Universal Robots URScript: SUB_107.script

def SUB_107():
  global _hidden_verificationVariable=0
  set_safety_mode_transition_hardness(1)
  set_tcp(p[0.0,0.09,0.42,0.0,0.0,0.0])
  set_target_payload(0.100000, [0.135000, 0.000000, 0.225000], [10.000000, 10.000000, 10.000000, 0.000000, 0.000000, 0.000000])
  set_gravity([0.0, 0.0, 9.82])
  set_standard_analog_input_domain(0, 1)
  set_standard_analog_input_domain(1, 1)
  set_tool_analog_input_domain(0, 1)
  set_tool_analog_input_domain(1, 1)
  set_analog_outputdomain(0, 0)
  set_analog_outputdomain(1, 0)
  set_input_actions_to_default()
  set_runstate_gp_boolean_output_to_value(0, 3)
  set_tool_communication(False, 115200, 0, 1, 1.5, 3.5)
  set_tool_output_mode(0)
  set_tool_digital_output_mode(0, 1)
  set_tool_digital_output_mode(1, 1)
  set_tool_voltage(0)
  global DistPillar=-0.10159
  global CandCnt=2
  global ReCaptZ=0.05
  global port=3000
  global socket_timeout=120
  global host="192.168.1.2"
  global is_popup=False
  global pBucket=[p[0.83653, 0.40397, 0.34225, 0, 0, -1.59904], p[-0.75609, -0.54132, 0.33714, 0, -0, 1.55997], p[0, 0, 0, 0, 0, 0]]
  global CaptStepZ=0.08
  global CaptIndex=[2, 0, 0]
  global pBucketM=p[-0.76064, -0.49997, 0.35503, 0, 0, 1.57135]
  global socket_name="vt"
  global rovi_err=0
  global SubPrgResult=100
  global CurrPos=p[-0.0041, -0.42062, 0.52846, -0.0222, -3.14131, -0.00178]
  global CurrPos_p=p[-0.00291, -0.33016, 0.10856, -0.0222, -3.14131, -0.00178]
  global ForceStartZ=0.39943
  global CutOffZ=0.26446
  global Sub3100_ZMax=0.74
  global ForceStartX=-0.90368
  global Sub3100_aRot=0.2
  global Sub3100_d=0.3
  global Sub3100_Option=38
  global Sub3100_a=0.2
  global Sub3100_XdV=0.1
  global Sub3100_XdRot=8
  global ZoneDistTh=0.05
  global BucketWidth=0.95
  global ZoneBucketGap=0
  global ZoneHomeX=0.2
  global UnloadZ=0.072
  global CaptPos=p[0.757, -0.42592, -0.06353, 3.14138, 0.03448, 0.00005]
  global BucketUpperPos=p[0.471, -0.42592, -0.06353, 3.14138, 0.03448, 0.00005]
  global Sub3100_GPII18=38
  global Zone6ThX=0.1
  global Zone6ThY=0.05
  global pCV=p[-0.00039, 0.00199, -0.01591, -0.0138, 0.00523, 0.00624]
  global CaptRowNo=5
  global CrankDepthFull=0.025
  global CrankDepth=0.12406
  global Y1=[2, -101.58556, 16.83588, 47.62585]
  global Y2=p[0.20537, -0.59585, -0.22377, -0.01856, -0.01958, 1.59883]
  global EvacRadiusTh=0.3
  global EvacXTh=[-0.5, 0.5]
  global EvacYTh=[-0.8, 1]
  global EvacZTh=[-0.1, 5]
  global WorkPosNo=0
  global Zone1ZTh=0.1
  global ReCaptNo=0
  global DistPillarBak=-0.10159
  global CaptIndexWk=2
  global PoseSub=p[0, 0, 0, -0.04215, -0.01806, 0]
  global PoseAdd=p[0.26591, -0.96698, -0.01503, 2.15596, 2.2396, -0.0019]
  global RZTh=15
  global pBucketC=p[0.45, -0.8, 0.35, 0, 0, 3.1415]
  global ReCaptZWk=0
  global CheckMST=1
  global RZSub=3.31201
  global DistPillarCOTh=0.16
  global DistPillarAPTh=0.26
  global CutOffZAdd=0.24763
  global CutOffZDef=0.09
  global Y8=0
  global BKWidth_Value=[934, 985, 0]
  global BKWidth_Name="/prepro/bucket_width"
  global LevelZ=0.01684
  global NeighborZ=0.04763
  global Currpos_p_UF0=p[0.27154, 0.19262, 0.33701, -2.25553, -2.16214, -0.02728]
  global TCPSpeed=p[0, 0, 0, 0, 0, 0]
  global Sub3100_Xd=[0, 0, -0.1, 0, 0, 0]
  global Sub3100_q=2
  global Sub3100_e=-1
  global Sub3100_t=0.5
  global IsShake=False
  global BeyondZ=0.2
  global ShakeCnt=-1
  global IsSteady_01=False
  global IsSteady_02=True
  global HandInZ=0.05
  global TCPSpeedThZ=0.0005
  global ShakeWaitSec=1
  global CutOffPos=p[0.74495, -0.05741, 0.23647, -2.14909, 2.29151, 0]
  global RelMoveZ=0.075
  global ForceFeature=p[0.83653, 0.40397, -0.05775, 0, 0, -1.59904]
  global ForceAxis=[1, 1, 1, 1, 1, 1]
  global ForceValue=[0, 0, -0.04, 0, 0, 0]
  global ForceType=2
  global ForceLimit=[0.01, 0.01, -0.02505, 0.17453, 0.17453, 0.17453]
  global ForceStep=3
  global IsBLLoad=False
  global TM_BLLoad=0.5
  global Sub104__TiltZTh=[0.25, 0.4]
  global Sub104_TiltZTh=[-0.5, 0.5]
  global BucketDef=p[0.83653, 0.40397, 0.34225, 0, 0, -1.59904]
  global ForceLimitZ=[0.015, 0.05, 0.05]
  global gGD_pos5=p[0.59447, 0.0126, 0.29998, 2.24881, -2.18946, -0.00407]
  global CutOffTCP=p[0, 0.09, 0.42, 0, 0, 0]
  global UseCutOffTCP=False
  global UseZSlide=False
  global UseBaseZRotate=True
  global BKWidth=0.942
  global Test01=1
  global CaptPointL_dX=0.185
  global CaptPointR_dX=0.185
  global UseShake=False
  global UseNewCaptPos=True
  global RZSupDegMin=[-5, 5]
  global RZSupForceVal=0
  global UseRZSuppress=True
  global TCPForce=p[-4.229, -4.99777, 6.44302, -0.65641, 0.21227, -0.12445]
  global TCPForceBak=p[-0.4161, 1.91403, -0.9967, 0.73001, 0.59984, -1.32957]
  global CVCorrDegMin=[-0.1, 0.1]
  global RZSupRatio=[1, 1]
  global RZSupOffset=[0, 0]
  global CVCorrRatio=[1.5, 1.5]
  global CVCorrOffset=[0, 0]
  global CVCorrRZVal=-1.55172
  global RYSub=-1.03448
  global UseCVCorr=True
  global RZSupForceRange=[-5, 5]
  global DistBKUpperTh=0.1
  global DistBKUpper=0.51791
  global StopSpeed=[0.005, 0.005, 0.005, 99999, 99999, 0.054]
  global RZSupRYRange=[-5, 5]
  global UseRZSupStep1=False
  global UseZRotate=False
  global CVCorrRYSub=-1.03448
  global CVCorrYVal=0.00758
  global DistOrigin=0.33017
  global v1=True
  global v2=True
  global v3=True
  global CVXTh=[-0.45, 0.45]
  global CVYTh=[-1, -0.7]
  global CVZTh=[-0.07, 5]
  global ForceVZDecay=0.04
  global ForceVZDecayWk=0.04
  global ForceLZDecay=0.00005
  global ForceLZDecayWk=0.00005
  global gGD_2_LM_Offset=p[0.001, 0, -0.00365, 0, 0, 0]
  global gGD_2_RM_Offset=p[0.0027, 0, -0.0018, 0, 0, 0]
  global ForceValueBak=[0, 0, 0, 0, 0]
  global TCPForceBak2=p[5.2035, -2.82194, -1.34504, -0.27224, -0.00796, -0.02911]
  global TCPSpeedBak2=p[0.01059, -0.00479, -0.01188, -0.01077, -0.06234, 0.02276]
  global gGD_2_LM_p=p[0.148, -0.5447, -0.0735, 0.248, 1.972, -2.179]
  global gGD_2_RM_p=p[0.1505, -0.54433, -0.069, 0.296, -2.013, 2.209]
  global gGD_2_M_p=p[0.149, -0.54489, -0.0725, -0.00488, 2.08628, -2.29812]
  global gGD_2_M_Offset=p[0.00149, 0, -0.00403, 0, 0, 0]
  global Bucket=p[0.32604,0.49174,0.0,-1.882900624652718E-5,2.8304179127934987E-5,-1.593185305749222]
  global BucketM=p[0.32604,0.49174,0.0,2.2353980716304163E-16,-3.5868426080024975E-16,-1.5931853071795856]
  global CV=p[0.0,0.0,0.0,0.0,0.0,0.0]
  global CaptPoint_C=p[-0.335,0.0,0.2915,-2.1962990605814006,-2.246289190961992,-5.664481053350347E-5]
  global CaptPoint_C2=p[0.32796661698047924,-0.010768520544682924,0.01931625281283378,2.2288103429550152,-2.213636886217198,8.598462540813273E-5]
  global CaptPoint_L=p[-0.335,-0.29,0.4,2.196198431950414,2.246349774520516,5.8693989933774055E-5]
  global CaptPoint_L2=p[0.327894307417917,-0.010799940826224014,0.01928712668893995,2.087717047309385,-2.0736781215133306,0.27365839887453103]
  global CaptPoint_R=p[-0.335,0.29,0.4,-2.1963472338807764,-2.2462285075856694,3.086531389441326E-5]
  global CaptPoint_R2=p[0.327926308680866,-0.010795166414457658,0.019300245403843563,-2.1186306375223185,2.1040550557443427,0.22023197678473694]
  global Capt_1BK_L=p[-0.395,-0.47,0.35,-2.1961210242572884,-2.2463362846055,-2.908274762447041E-4]
  global Capt_1BK_R=p[-0.395,0.51,0.35,2.196067754706757,2.246288285862388,2.8411291050601595E-5]
  global Capt_1BK_pos1=p[-0.4218793038724447,-0.003154429464978058,0.2915499891144615,-2.1963422029204875,-2.2438663520270015,-0.02197160668673838]
  global Capt_1BK_pos2=p[-0.42187829024618434,-0.0031710253373066375,0.29156503858953065,-2.196324918349679,-2.2439040699490773,-0.021928444416953782]
  global Capt_2BK_L=p[0.42186661528427194,0.4254738068040517,0.35042275762909847,2.239156309475874,-2.1837044610999294,0.002643817066643282]
  global Capt_2BK_R=p[0.4218208572756906,-0.5427676723257963,0.350372239919558,2.2392697861179327,-2.183553596194912,0.002410470905346486]
  global Capt_2BK_pos1=p[0.42193501458435656,0.004742683868356356,0.35045865974037793,2.2391012408536453,-2.1839704655717003,0.002677867056024068]
  global Capt_2BK_pos2=p[0.421903984494575,0.004707988774967922,0.35045218900915065,2.239114367170047,-2.183895515396197,0.002684056681074047]
  global Capt_CV_M=p[-0.04794223960540197,-0.559868557160475,0.1086937653706071,-0.022464429848058916,-3.141454018347238,4.0166993855964835E-4]
  global Capt_GD_M=p[-0.004053197679954899,-0.25261725691632436,-0.01970497430780127,0.0332779454553888,-3.140179196376707,-0.0034093680964018282]
  global HomePointL=p[-0.36789,-0.5117344641471838,0.78,-0.6278857271586024,3.0680899128661667,-8.649957362498864E-4]
  global Master_pos=p[0.121,-0.17,-0.0545,-0.020993616946531908,-3.141044973619201,0.0]
  global Master_posL=p[-0.003,-0.27,0.109,0.02094395102393583,3.0543261909900803,-5.235987755386035E-4]
  global Master_posR=p[-0.003,-0.27,0.109,-0.019810987664379186,-3.054193931591229,4.952746915529204E-4]
  global Master_pos_1=p[0.11094339812903395,-0.23710672065782984,0.08047378202276018,-0.05666752666458696,3.1228966394147033,0.01312068089365201]
  global PickPos=p[0.10830682331105715,-1.3709505888096256,-0.18404188875951455,-0.00622194000158997,2.880236948927292,-0.00383636509397631]
  global Solve=p[-0.00368,-0.0021000000000000003,0.25739999999999996,0.0,0.0,0.0]
  global TCP3100TL=p[0.0,0.08,0.42,1.8939999999999997,0.0,0.0]
  global TEST=p[0.1,0.0,0.2,0.0,0.0,0.0]
  global TEST_ROTSUP=p[-0.07293017509777999,-0.3201239472424659,0.14015840016860298,-0.014967413338418362,-3.108805898474534,-0.035972414862118114]
  global UF=p[0.0,0.0,0.0,0.0,0.0,0.0]
  global g1CV_posL1=p[0.05028133628211688,-0.4526481033729615,0.1221845548632916,-2.213335080948508,-2.1937561336067057,-0.3280056759040735]
  global g1CV_posR1=p[0.03743870476062511,-0.53119407812668,0.11301901343688614,2.073418671558482,2.153257467049566,0.11656306439039889]
  global g1GD_pos1=p[0.15518019183109402,-0.6360044329537242,0.2714505325043806,2.2006040244311444,2.21554807672813,0.0172874948472804]
  global g1GD_pos2=p[0.03949427043618803,-0.46718749500887935,0.4516738215011898,2.194658091359525,2.207226449099828,0.02874313290876032]
  global g1GD_pos3=p[-0.18905837741804024,-0.43030396733112375,0.45070429849649235,2.659275306106194,1.6146847883250424,0.011588789466751665]
  global g1GD_pos4=p[-0.25628841794770224,-0.020630481098425146,0.45,2.148716725221303,2.2918109407224354,-1.3854918368741778E-5]
  global g1GD_pos5=p[-0.7020222150975298,-0.020008703038085586,0.44884773524121807,2.130900859862887,2.274424413859522,0.03157573215401506]
  global g1GD_pos5_NEAR=p[-0.5143300000000001,-0.023002183632447833,0.4499678963159493,2.1476150413314157,2.292837734093618,6.185870865614646E-5]
  global g1GD_posL1=p[-0.08276848269606216,-0.3996147100031649,0.1488453551331823,2.286527078917204,1.8420745504477611,0.33698451773695576]
  global g1GD_posL2=p[-0.3253977027403738,-0.3024804624281039,0.16332814085945146,2.72312820760317,0.9631021078169197,0.32447452035226126]
  global g1GD_posL3=p[-0.6791033397183219,0.06787475590683856,0.16337212788108813,2.1383125299263996,2.086116032377724,0.4536080263755059]
  global g1GD_posR1=p[-0.09893370538053747,-0.4999608954567234,0.14329885217724153,2.43311852414254,1.4238397520832589,0.08559216753941556]
  global g1GD_posR2=p[-0.3729565201882258,-0.3752983669473301,0.143299052800563,2.6951655216297596,0.8130506811102118,-0.02387549506099888]
  global g1GD_posR3=p[-0.7385929502572233,-0.029472684480355026,0.1499650660949685,2.0484522752014467,1.9493695704119496,0.18368227556562683]
  global g2CV_posL1=p[0.3409386496330911,-0.4656338066361442,0.1250074988128972,2.209372209162659,2.1945371304665926,0.3160714960040194]
  global g2CV_posR1=p[0.3400736278759575,-0.531334269888987,0.1183415684753657,2.07314649492589,2.1532617466521136,0.11638666128062146]
  global g2GD_pos1=p[0.2541388115968006,-0.677503610088671,0.18526502532787942,-2.037688671369965,-2.388999479520465,-0.002109631087665523]
  global g2GD_pos2=p[0.26549608295016686,-0.43417144272655195,0.3031020231265486,1.8657349645042864,2.5176803321572097,0.03468085036703408]
  global g2GD_pos3=p[0.33816249037197144,-0.05647845608560481,0.3023625116884547,-0.13692892188304248,3.136351554782643,0.02916083337488691]
  global g2GD_pos4=p[0.31242512329230154,0.14446123595746882,0.30198009989558844,1.0729609473784474,-2.951947119809616,-0.018083971938859904]
  global g2GD_pos5=p[0.5944722301546509,0.012599499854360038,0.29997637895993046,2.2488051716265702,-2.189457282897882,-0.004073585227441316]
  global g2GD_pos5_NEAR=p[0.5968300000000001,0.0128,0.44997000000000004,2.250000000000808,-2.1920000000007867,0.0]
  global gCV_11_M=p[0.2915530857570407,-0.971,-0.025,2.1278112861740515,2.1191563150105255,0.2692956395397443]
  global gCV_12_M=p[0.345821498078164,-0.971,-0.025,2.1151831254696565,2.1296350097775147,0.29070323755963534]
  global gCV_13_M=p[0.3651558412628,-0.8681469245134871,0.07328969396678225,2.1152334618409543,2.1295870661800307,0.2908325984974855]
  global gCV_1_M=p[0.26591000000000004,-0.9669777782584144,-0.015030098319161023,2.186106464667012,2.2102154916004255,-0.0025904121924328924]
  global gCV_2_M=p[0.26591000000000004,-0.9669800000000001,0.0368486796934106,2.1889216892500283,2.199870474563767,0.009420192863142347]
  global gCV_3_M=p[0.29099390607376485,-0.6570558385379063,0.0722153583041818,1.9884242634571576,2.2321538498123994,0.15249643504377583]
  global gCV_pos5=p[0.3400172856834047,-0.9722754606605235,-0.18287928563575456,2.073394561413637,2.1531827558666565,0.11639000988241816]
  global gGD_1_LM=p[0.02419,-0.7289500000000001,-0.11494,-0.010169347158913017,2.870767181856166,0.2884627079222753]
  global gGD_1_LM_RX=p[0.02416,-0.7290503881876362,-0.11492000000000001,0.3044368416109271,1.9674275598429376,-2.2260150226690767]
  global gGD_1_LM_RXF=p[0.02413503458160308,-0.74534,-0.11578000000000001,0.2411332216392182,1.7407173006243832,-2.3674279033231747]
  global gGD_1_M=p[0.023469999999999998,-0.72661,-0.11456000000000001,-0.029570847824802682,-3.12419917405015,-0.3106340785404749]
  global gGD_1_M_RX=p[0.023469999999999998,-0.7267389086136226,-0.11653,-0.01497665825746678,-2.067091763806016,2.343829767295237]
  global gGD_1_M_RXF=p[0.02415523713330076,-0.7453200000000001,-0.11578426509069895,-0.012477314995716382,-1.853515977408631,2.515027308648709]
  global gGD_1_RM=p[0.023629999999999998,-0.72653,-0.11331000000000001,-0.06253229749015264,-2.8808212567082414,-0.28238046714011755]
  global gGD_1_RM_RX=p[0.023710000000000002,-0.7266791760279572,-0.11328,0.25928042729790574,-1.9492131299374433,2.2165015837642534]
  global gGD_1_RM_RXF=p[0.024158234647744328,-0.74536,-0.11577,0.21548497967238725,-1.726437707763004,2.3373117534316665]
  global gGD_2_LM=p[0.02467,-0.67055,-0.11509,-0.010179461791212513,2.870955921048522,0.2878734195391217]
  global gGD_2_LM_RX=p[0.147,-0.5447000000000001,-0.06985,0.24799999999999686,1.9720000000000022,-2.179000000000001]
  global gGD_2_LM_RXF=p[0.02518,-0.6822999999999999,-0.11982,0.24121310672797797,1.7407223643292684,-2.3672997334921986]
  global gGD_2_M=p[0.02389,-0.6721900000000001,-0.11456000000000001,-0.029666521928107308,-3.1243201149134068,-0.3098990972493868]
  global gGD_2_M_RX=p[0.14751,-0.54489,-0.06847,-0.0048813183873774365,2.0862754787651414,-2.298124696777323]
  global gGD_2_M_RXF=p[0.02469,-0.68228,-0.11781,-0.012625584579695818,-1.8536977166603092,2.514979910589354]
  global gGD_2_RM=p[0.02429,-0.66916,-0.11353,-0.06253008389277029,-2.880917079483223,-0.28230802316028863]
  global gGD_2_RM_RX=p[0.14780000000000001,-0.5443300000000001,-0.06720000000000001,0.2959999999999995,-2.0130000000000017,2.209000000000002]
  global gGD_2_RM_RXF=p[0.02418,-0.68221,-0.11985,0.21545635593876583,-1.7267658137434814,2.337110041109278]
  global gGD_3_LM=p[0.024149999999999998,-0.63442,-0.00372,-0.010168641563882792,2.8709293839329573,0.28786844960240987]
  global gGD_3_LM_RX=p[0.14789,-0.51554,-0.06981,0.24799999999999944,1.9709999999999999,-2.1789999999999994]
  global gGD_3_LM_RXF=p[0.02387752228160463,-0.5964211774687285,-0.05792315514989682,0.2704410553277331,1.9481847980902196,-2.214876983085744]
  global gGD_3_M=p[0.023940000000000003,-0.63613,-0.00522,-0.029962916255114207,-3.1241595671421933,-0.3100480455299553]
  global gGD_3_M_RX=p[0.14743,-0.51525,-0.06848,-0.004881318387378877,2.086275478765143,-2.2981246967773257]
  global gGD_3_M_RXF=p[0.02383447419609676,-0.5964085561522618,-0.0579509198373786,-0.014600929068906539,-2.066655165579624,2.3438719244209403]
  global gGD_3_RM=p[0.02428,-0.6347200000000001,-0.00846,-0.0624152449577923,-2.8809080008278345,-0.2823877130468296]
  global gGD_3_RM_RX=p[0.14778,-0.5151,-0.06720000000000001,0.2959999999999995,-2.0130000000000017,2.209000000000002]
  global gGD_3_RM_RXF=p[0.023773322279514588,-0.5964087734876792,-0.05795139315103717,0.24060086319727583,-1.933030903056379,2.187075285864524]
  global gGD_4_LM=p[-0.011210304327025133,-0.5154273285739928,0.03,0.24806379354211447,1.9716743582538676,-2.178783821422816]
  global gGD_4_LM_RX=p[-0.12533199352487323,-0.6346108123799734,-0.003643920282847657,0.304552460658092,1.9670859988240124,-2.226395027960848]
  global gGD_4_RM=p[0.30796717945535684,-0.5151064262102534,0.03,0.29563155154414866,-2.013445679592415,2.2089997240372727]
  global gHome_Position=p[-0.0028799999999999997,-0.33081,0.1087,-0.02099958342773921,-3.141491282453575,3.986162810876369E-4]
  global gTAIHI_pos1=p[0.034435296708333146,-0.2890869270984411,0.28697762766096685,-0.9517096680276043,2.9907327255336362,-0.006242657270483182]
  global gTAIHI_pos2=p[0.46041690381401934,0.09562026346103787,0.3409455343940188,-2.575428180750575,1.7504967205574518,-0.009370784990557466]
  global gTAIHI_pos3=p[0.4777514786587304,0.10855417509450788,0.25667938190447326,-3.115092130529677,-0.059113053813058626,0.017060902648732133]
  global gTAIHI_pos4=p[0.47773948064032057,0.10853581553326999,-0.15133852019421468,-3.1151611852917296,-0.05914313994407087,0.017149581050184888]
  global gTAIHI_pos5=p[0.30588450070104545,0.17870028478253597,-0.38750721344025674,-3.115302721311487,-0.05927431563397507,0.01725874757592571]
  global p0507=p[-0.335,0.29,0.4,-2.152,-2.1999999999999993,-0.09000000000000297]
  rtde_set_watchdog("speed_slider_mask", 10.0, "ignore")
  # begin: URCap Installation Node
  #   Source: Ethernet/IP I/O Monitor URCap, 1.0.0,
  #   Type: Ethernet/IP I/O Monitor
  conn = rpc_factory("xmlrpc", "http://127.0.0.1:" + to_str(61101) + "/RPC2")

  def show_monitor():
    return conn.eip_monitor.show()
  end
  # end: URCap Installation Node
  step_count_fb5cdaa9_2a23_499d_bf21_999fa2243354 = 0.0
  thread Step_Counter_Thread_2a7e4f0a_567e_4262_afd5_7eee6c683445():
    while (True):
      step_count_fb5cdaa9_2a23_499d_bf21_999fa2243354 = step_count_fb5cdaa9_2a23_499d_bf21_999fa2243354 + 1.0
      sync()
    end
  end
  run Step_Counter_Thread_2a7e4f0a_567e_4262_afd5_7eee6c683445()
  while (True):
    $ 2 "ロボットプログラム"
    $ 3 "FREE_DRIVE"
    $ 4 "freedrive_mode()"
    freedrive_mode()
    $ 5 "荷重の設定: k2"
    set_target_payload(0.100000, [0.135000, 0.000000, 0.225000], [2.000000, 2.000000, 2.000000, 0.000000, 0.000000, 0.000000])
    $ 6 "設定"
    set_tcp(p[0.0,0.0,0.0,0.0,0.0,0.0])
    $ 7 "待機: 1.0"
    sleep(1.0)
    $ 8 "end_freedrive_mode()"
    end_freedrive_mode()
    $ 9 "CV_CORR_RZ"
    $ 10 "If文 UseCVCorr"
    if (UseCVCorr):
      $ 11 "設定"
      set_tcp(p[0.0,0.09,0.42,0.0,0.0,0.0])
      $ 12 "sync()"
      sync()
      $ 13 "CurrPos_p=get_actual_tcp_pose()"
      CurrPos_p= get_actual_tcp_pose ()
      $ 14 "CurrposAligned:=p[0,0,0,0,0,0]"
      global CurrposAligned=p[0,0,0,0,0,0]
      $ 15 "CurrposAligned:=GET_ALIGNED_TCP(CurrposAligned)"
      global CurrposAligned=GET_ALIGNED_TCP(CurrposAligned)
      $ 16 "GET_CVCORR_VALUE(CurrposAligned)"
      GET_CVCORR_VALUE(CurrposAligned)
    end
  end
end
